TYPE ST_EP9224_SlaveOut :
STRUCT
	nChannel :ARRAY [1..EP9224_NUM_CHANNELS] OF BYTE;
	nStatus	 :BYTE;
END_STRUCT
END_TYPE

(* stored: Version 1.1.0.1, ProductVersion 3.1.4024.9
   DUT ST_EP9224_SlaveOut: Id {26189417-0e45-45b9-8132-d598dbceae69} *)
